(* CODESYS project UDP.GPRS.200205.02.project

Project tree, tasks and I/O mapping:
  Device : Changsha-Cyber-MI-linux, Changsha Cyber-MI Co., Ltd., version 3.5.10.40
    application Application
      libraries: Standard, * (System); SysFile, 3.5.15.0 (System); SysTypes2 Interfaces, * (System); SysShm, * (System); CAA Mathematics, * (CAA Technical Workgroup); SysTime, 3.5.9.0 (System); CAA Types Extern, 3.5.13.0 (CAA Technical Workgroup); TCP, 3.5.15.0 (3S - Smart Software Solutions GmbH); CAA Net Base Services, 3.5.15.0 (CAA Technical Workgroup)
      task c_MainTask (cyclic, interval 10 ms, priority 20) calls prg_main
      data type STATE
      programs/
        program prg_main [ST]
    SoftMotion General Axis Pool
  libraries: VisuSymbols, 3.5.10.0 (System)
  5ce3da45-db07-42e7-a21c-a00fff4ed8f6|C:\Users\zhou\p01.bmp
  5ce3da45-db07-42e7-a21c-a00fff4ed8f6|C:\working\p01.bmp
  5ce3da45-db07-42e7-a21c-a00fff4ed8f6|C:\working\file.bmp
  text list GlobalTextList
*)

// Device/Application/STATE
TYPE STATE :
(
	INIT := 0, 	(* first State. Connections are set up *)
	SEND,		(* Send messages *)
	READ,		(* Receive messages *)
	ERROR		(* Prepare to reset connections *)
);
END_TYPE

// Device/Application/programs/prg_main
PROGRAM prg_main
VAR  
	eSTATE			: STATE; (* 状态转换变量 *)
	
	myIP		: NBS.IP_ADDR; (* MIC7001本身的IP地址 *)
	myPort		: UINT; (* MIC7001用于通信的端口 *)
	IPSend		: NBS.IP_ADDR; (* 对方的IP地址 *)
	PortSend	: UINT; (* 对方的端口 *)

	sToSend			: STRING; (* 待发送数据 *)
	sReceived		: STRING; (* 接收数据 *)

	ctRecAnswers	: CAA.COUNT; (* No. of received messages *)
	ctSentMessage	: CAA.COUNT; (* No. of sent messages *)
	ctErrorCounter	: CAA.COUNT; (* No. connection errors *)

	UDPPeer			: NBS.UDP_Peer; (* FB UDP Peer *)
	UDPSend			: NBS.UDP_Send; (* FB UDP Send *)
	UDPReceive		: NBS.UDP_Receive; (* FB UDP Receive *)
	
	Peer			: CAA.HANDLE; (* Handle to the peer connection *)
	
	/// 辅助变量 
	xSend			: BOOL;
	i				: UINT;
	sTmp1			: STRING;
	xEnable			: BOOL;
	
END_VAR


CASE eSTATE OF

STATE.INIT:  //初始化状态
	myIP.sAddr:= '0.0.0.0';	
	myPort:= 8888;
	
	sToSend:= 'Hello World: ';
	xEnable:= TRUE;  //用于启动最下方的第70行的UDPPeer
	// 建立连接后马上转到发送状态
	IF UDPPeer.xActive THEN 
		eSTATE:= STATE.send;
	ELSIF UDPPeer.xError THEN
		eSTATE:= STATE.ERROR;
	END_IF
		
STATE.SEND:  //发送状态
	//发送一个字符串加一个数字（100到0）
	IF UDPPeer.xActive THEN 
		xSend:= TRUE;
		IF i = 0 THEN
			i:= 100;
		END_IF
	
		sTmp1 := concat(STR1 := sToSend, STR2 := UINT_TO_STRING(i));
		sTmp1 := concat(STR1 := sTmp1, STR2 := '$r');
		IPSend.sAddr := '47.107.240.29';	
		PortSend := 23457;
		UDPSend(xExecute:= xSend, udiTimeOut:= 0, hPeer:= Peer, ipAddr:= IPSend, uiPort:= PortSend, szSize:= len(sTmp1), pData:= ADR(sTmp1));
		//发送成功后发送的数字减一，并转入接收状态
		IF UDPSend.xDone THEN 
			i:= i -1;				
			UDPSend(xExecute:= FALSE);	
			xSend:= FALSE;
			ctSentMessage:= ctSentMessage +1;
		
			eSTATE:= STATE.read;
		ELSIF UDPSend.xError THEN
			eSTATE:= STATE.ERROR;		
		END_IF
	ELSE
		eSTATE:= STATE.ERROR;
	END_IF
	

STATE.READ:  //接收状态
	//如果收到数据，则转入发送状态，发送下一帧
	//如果出现错误，进入错误状态
	IF UDPPeer.xActive THEN 
		sReceived := '';
		UDPReceive(xEnable:= TRUE,  hPeer:= Peer, szSize:= SIZEOF(sReceived), pData:= ADR(sReceived));
		IF UDPReceive.xReady THEN
			ctRecAnswers:= ctRecAnswers +1;
			eSTATE:= STATE.SEND;
		ELSIF UDPReceive.xError THEN
			eSTATE:= STATE.ERROR;
		END_IF
	ELSE
		eSTATE:= STATE.ERROR;
	END_IF
	
STATE.ERROR:  //错误状态
	ctErrorCounter:= ctErrorCounter +1;
	xEnable := FALSE;
	eState := STATE.INIT;	 //回到初始化状态，重新开始

END_CASE

//保持每个周期调用，维护与对方的连接关系本地端口的接收状态
UDPPeer(xEnable:= xEnable, ipAddr:= myIP, uiPort:= myPort, hPeer=> Peer);

END_PROGRAM
